// SIMATIC STEP 7 (V5.x) project Put_Get
// CPU: CPU 414-5 H (ATC-RSM)
// CPU: CPU 414-5 H (OPC-OA)
// station: P_ADR_BUS
// station: Hardware
// station: SIMATIC 400(ATC-RSM)
// station: SIMATIC 400(OPC-OA)
// station: P_ADR_BUS
// station: Hardware
// program: S7 Program
// program: S7 Program(1)

SYMBOL_TABLE
"Receive_DB"	DB 50	DB 50
"Send_DB"	DB 51	DB 51
"GET_DB"	DB 52	SFB 14
"PUT_DB"	DB 53	SFB 15
"CPU_Comm"	FC 1	FC 1
"CPU_Communication"	FC 199	FC 199
"ASSAP"	I 0.0	BOOL	//  (ATC) - (FieldIO4-M1)
"BOPL"	I 0.1	BOOL	//  (ATC) - (FieldIO4-M1)
"BVAP"	I 0.2	BOOL	//  (ATC) - (FieldIO4-M1)
"DVSAP"	I 0.3	BOOL	//  (ATC) - (FieldIO4-M1)
"EHFPL"	I 0.4	BOOL	//  (ATC) - (FieldIO4-M1)
"EHSO"	I 0.5	BOOL	//  (ATC) - (FieldIO4-M1)
"GDOGF"	I 0.6	BOOL	//  (ATC) - (FieldIO4-M1)
"GVRNLV"	I 0.7	BOOL	//  (ATC) - (FieldIO4-M1)
"HPDVC"	I 1.0	BOOL	//  (ATC) - (FieldIO4-M1)
"HPDVO"	I 1.1	BOOL	//  (ATC) - (FieldIO4-M1)
"MBCSU"	I 1.2	BOOL	//  (ATC) - (FieldIO4-M1)
"MELIT"	I 1.3	BOOL	//  (ATC) - (FieldIO4-M1)
"MVHPIT"	I 1.4	BOOL	//  (ATC) - (FieldIO4-M1)
"OEPIT"	I 1.5	BOOL	//  (ATC) - (FieldIO4-M1)
"RSBC"	I 1.6	BOOL	//  (ATC) - (FieldIO4-M1)
"RSBSU"	I 1.7	BOOL	//  (ATC) - (FieldIO4-M1)
"TGE"	I 2.0	BOOL	//  (ATC) - (FieldIO5-M1)
"VRO"	I 2.1	BOOL	//  (ATC) - (FieldIO5-M1)
"VROUS"	I 2.2	BOOL	//  (ATC) - (FieldIO5-M1)
"VRSOTP"	I 2.3	BOOL	//  (ATC) - (FieldIO5-M1)
"CAB4T1"	IW 512	WORD	//  (RSM) - (FieldIO4-M3)
"CNDP1"	IW 514	WORD	//  (RSM) - (FieldIO4-M3)
"FSST1"	IW 516	WORD	//  (RSM) - (FieldIO4-M3)
"B1T1"	IW 518	WORD	//  (ATC) - (FieldIO4-M3)
"B2T1"	IW 520	WORD	//  (ATC) - (FieldIO4-M3)
"B3T1"	IW 522	WORD	//  (ATC) - (FieldIO4-M3)
"B4T1"	IW 524	WORD	//  (ATC) - (FieldIO4-M3)
"B5T1"	IW 526	WORD	//  (ATC) - (FieldIO4-M3)
"B6T1"	IW 528	WORD	//  (ATC) - (FieldIO4-M4)
"RP1"	IW 530	WORD	//  (ATC) - (FieldIO4-M4)
"TBFCT1"	IW 532	WORD	//  (ATC) - (FieldIO4-M4)
"TBFLT1"	IW 534	WORD	//  (ATC) - (FieldIO4-M4)
"TBRCT1"	IW 536	WORD	//  (ATC) - (FieldIO4-M4)
"TBRLT1"	IW 538	WORD	//  (ATC) - (FieldIO4-M4)
"VB9"	IW 540	WORD	//  (ATC) - (FieldIO4-M4)
"FSMT1"	IW 542	WORD	//  (RSM) - (FieldIO4-M4)
"B7T"	IW 544	WORD	//  (ATC) - (FieldIO4-M5)
"B8T"	IW 546	WORD	//  (ATC) - (FieldIO4-M5)
"B9T"	IW 548	WORD	//  (ATC) - (FieldIO4-M5)
"B10T"	IW 550	WORD	//  (ATC) - (FieldIO4-M5)
"CAB5T1"	IW 552	WORD	//  (ATC) - (FieldIO4-M5)
"CAB5T2"	IW 554	WORD	//  (ATC) - (FieldIO4-M5)
"CASEXP"	IW 556	WORD	//  (ATC) - (FieldIO4-M5)
"DEGEN"	IW 558	WORD	//  (ATC) - (FieldIO4-M5)
"VB1"	IW 560	WORD	//  (ATC) - (FieldIO4-M6)
"VB2"	IW 562	WORD	//  (ATC) - (FieldIO4-M6)
"VB3"	IW 564	WORD	//  (ATC) - (FieldIO4-M6)
"VB4"	IW 566	WORD	//  (ATC) - (FieldIO4-M6)
"VB5"	IW 568	WORD	//  (ATC) - (FieldIO4-M6)
"VB6"	IW 570	WORD	//  (ATC) - (FieldIO4-M6)
"VB7"	IW 572	WORD	//  (ATC) - (FieldIO4-M6)
"VB8"	IW 574	WORD	//  (ATC) - (FieldIO4-M6)
"CAB4T2"	IW 576	WORD	//  (RSM) - (FieldIO5-M3)
"CNDP2"	IW 578	WORD	//  (RSM) - (FieldIO5-M3)
"FSST2"	IW 580	WORD	//  (RSM) - (FieldIO5-M3)
"B1T2"	IW 582	WORD	//  (ATC) - (FieldIO5-M3)
"B2T2"	IW 584	WORD	//  (ATC) - (FieldIO5-M3)
"B3T2"	IW 586	WORD	//  (ATC) - (FieldIO5-M3)
"B4T2"	IW 588	WORD	//  (ATC) - (FieldIO5-M3)
"B5T2"	IW 590	WORD	//  (ATC) - (FieldIO5-M3)
"B6T2"	IW 592	WORD	//  (ATC) - (FieldIO5-M4)
"RP2"	IW 594	WORD	//  (ATC) - (FieldIO5-M4)
"TBFCT2"	IW 596	WORD	//  (ATC) - (FieldIO5-M4)
"TBFLT2"	IW 598	WORD	//  (ATC) - (FieldIO5-M4)
"TBRCT2"	IW 600	WORD	//  (ATC) - (FieldIO5-M4)
"TBRLT2"	IW 602	WORD	//  (ATC) - (FieldIO5-M4)
"VB10"	IW 604	WORD	//  (ATC) - (FieldIO5-M4)
"LPGST"	IW 606	WORD	//  (RSM) - (FieldIO5-M4)
"EHFLT"	IW 608	WORD	//  (ATC) - (FieldIO5-M5)
"HPBMIDT"	IW 610	WORD	//  (ATC) - (FieldIO5-M5)
"HPCMIDT"	IW 612	WORD	//  (ATC) - (FieldIO5-M5)
"LP1GNT"	IW 614	WORD	//  (ATC) - (FieldIO5-M5)
"LP1GVT"	IW 616	WORD	//  (ATC) - (FieldIO5-M5)
"LP2GNT"	IW 618	WORD	//  (ATC) - (FieldIO5-M5)
"LP2GVT"	IW 620	WORD	//  (ATC) - (FieldIO5-M5)
"ROTECC"	IW 622	WORD	//  (ATC) - (FieldIO5-M5)
"OCIT"	IW 624	WORD	//  (RSM) - (FieldIO5-M6)
"OCOT"	IW 626	WORD	//  (RSM) - (FieldIO5-M6)
"Main Routine"	OB 1	OB 1
"OBNL_FLT"	OB 85	OB 85	// OB Not Loaded Fault
"PROG_ERR"	OB 121	OB 121	// Programming Error
"MOD_ERR"	OB 122	OB 122	// Module Access Error
"ATCALO"	Q 0.0	BOOL	//  (ATC) - (FieldIO4-M2)
"ATCASSO"	Q 0.1	BOOL	//  (ATC) - (FieldIO4-M2)
"ATCMEO"	Q 0.2	BOOL	//  (ATC) - (FieldIO4-M2)
"ATCNAO"	Q 0.3	BOOL	//  (ATC) - (FieldIO4-M2)
"ATCSMO"	Q 0.4	BOOL	//  (ATC) - (FieldIO4-M2)
"ATCTAO"	Q 0.5	BOOL	//  (ATC) - (FieldIO4-M2)
"ATCTO"	Q 0.6	BOOL	//  (ATC) - (FieldIO4-M2)
"CHPDVO"	Q 0.7	BOOL	//  (ATC) - (FieldIO4-M2)
"CRSBO"	Q 1.0	BOOL	//  (ATC) - (FieldIO4-M2)
"LPHTO"	Q 1.1	BOOL	//  (ATC) - (FieldIO4-M2)
"LPVHTO"	Q 1.2	BOOL	//  (ATC) - (FieldIO4-M2)
"WDHTO"	Q 1.3	BOOL	//  (ATC) - (FieldIO4-M2)
"WDVHTO"	Q 1.4	BOOL	//  (ATC) - (FieldIO4-M2)
"RSINV1"	Q 2.0	BOOL	//  (RSM) - (FieldIO5-M2)
"RSINV2"	Q 2.1	BOOL	//  (RSM) - (FieldIO5-M2)
"RSMON1"	Q 2.2	BOOL	//  (RSM) - (FieldIO5-M2)
"RSMON2"	Q 2.3	BOOL	//  (RSM) - (FieldIO5-M2)
"RSSENO"	Q 2.4	BOOL	//  (RSM) - (FieldIO5-M2)
"SPHLD"	Q 2.5	BOOL	//  (RSM) - (FieldIO5-M2)
"VAT (ATC-RSM)"	VAT 1	
END_SYMBOL_TABLE

FUNCTION "CPU_Communication" : VOID	// FC 199
TITLE = CPU_Comm
//Function call to read and write the CPU data
//
VERSION : 0.1
BEGIN
NETWORK
TITLE = Recieve data
      A     DB1.DBX 0.0;
      =     L 0.0;
      BLD   103;
      BLD   9;
      =     L 5.0;
      CDB;
      OPN   DI 1;
      TAR2  LD 1;
      A     L 0.0;
      =     DIX 0.0;
      L     1;
      T     DIW 2;
      L     W#16#1001;
      T     DIW 8;
      L     1;
      T     DIW 10;
      L     0;
      T     DIW 12;
      L     P#M 10.1;
      T     DID 14;
      L     W#16#1004;
      T     DIW 18;
      L     1;
      T     DIW 20;
      L     0;
      T     DIW 22;
      L     P#M 11.0;
      T     DID 24;
      L     W#16#1006;
      T     DIW 28;
      L     1;
      T     DIW 30;
      L     0;
      T     DIW 32;
      L     P#M 13.0;
      T     DID 34;
      L     W#16#1004;
      T     DIW 38;
      L     1;
      T     DIW 40;
      L     0;
      T     DIW 42;
      L     P#M 17.0;
      T     DID 44;
      L     W#16#1001;
      T     DIW 48;
      L     1;
      T     DIW 50;
      L     0;
      T     DIW 52;
      L     P#M 0.1;
      T     DID 54;
      L     W#16#1005;
      T     DIW 58;
      L     1;
      T     DIW 60;
      L     0;
      T     DIW 62;
      L     P#M 1.0;
      T     DID 64;
      L     W#16#1008;
      T     DIW 68;
      L     1;
      T     DIW 70;
      L     0;
      T     DIW 72;
      L     P#M 3.0;
      T     DID 74;
      L     W#16#1004;
      T     DIW 78;
      L     1;
      T     DIW 80;
      L     0;
      T     DIW 82;
      L     P#M 7.0;
      T     DID 84;
      LAR2  P#DBX 0.0;
      UC    SFB 14;
      LAR2  LD 1;
      A     DIX 4.0;
      OPN   DI 1;
      =     DIX 4.0;
      OPN   DI 1;
      A     DIX 4.1;
      OPN   DI 1;
      =     DIX 4.1;
      OPN   DI 1;
      L     DIW 6;
      OPN   DI 1;
      T     DIW 6;
      OPN   DI 1;
      CDB;
      BLD   10;
      NOP   0;
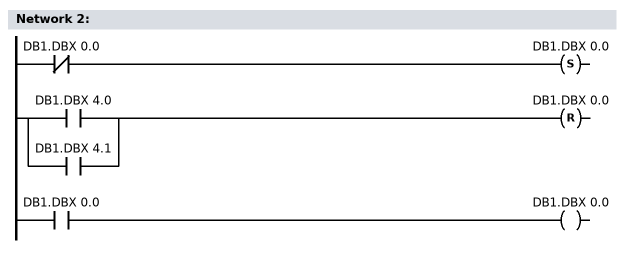
NETWORK
TITLE =
      AN    DB1.DBX 0.0;
      S     DB1.DBX 0.0;
      A(;
      O     DB1.DBX 4.0;
      O     DB1.DBX 4.1;
      );
      R     DB1.DBX 0.0;
      A     DB1.DBX 0.0;
      =     DB1.DBX 0.0;
END_FUNCTION

DATA_BLOCK "Receive_DB"	// DB 50
VERSION : 0.1
  STRUCT
   DB_VAR : INT ;	//Temporary placeholder variable
  END_STRUCT ;	
BEGIN
END_DATA_BLOCK

DATA_BLOCK "Send_DB"	// DB 51
VERSION : 0.1
  STRUCT
   DB_VAR : INT ;	//Temporary placeholder variable
  END_STRUCT ;	
BEGIN
END_DATA_BLOCK

DATA_BLOCK "GET_DB"	// DB 52
AUTHOR : SIMATIC
FAMILY : COM_FUNC
VERSION : 0.1
SFB 14
BEGIN
END_DATA_BLOCK

DATA_BLOCK "PUT_DB"	// DB 53
AUTHOR : SIMATIC
FAMILY : COM_FUNC
VERSION : 0.1
SFB 15
BEGIN
END_DATA_BLOCK

ORGANIZATION_BLOCK "Main Routine"	// OB 1
TITLE = "Main Program Sweep (Cycle)"
VERSION : 0.1
VAR_TEMP
  OB1_EV_CLASS : BYTE ;	//Bits 0-3 = 1 (Coming event), Bits 4-7 = 1 (Event class 1)
  OB1_SCAN_1 : BYTE ;	//1 (Cold restart scan 1 of OB 1), 3 (Scan 2-n of OB 1)
  OB1_PRIORITY : BYTE ;	//Priority of OB Execution
  OB1_OB_NUMBR : BYTE ;	//1 (Organization block 1, OB1)
  OB1_RESERVED_1 : BYTE ;	//Reserved for system
  OB1_RESERVED_2 : BYTE ;	//Reserved for system
  OB1_PREV_CYCLE : INT ;	//Cycle time of previous OB1 scan (milliseconds)
  OB1_MIN_CYCLE : INT ;	//Minimum cycle time of OB1 (milliseconds)
  OB1_MAX_CYCLE : INT ;	//Maximum cycle time of OB1 (milliseconds)
  OB1_DATE_TIME : DATE_AND_TIME ;	//Date and time OB1 started
END_VAR
BEGIN
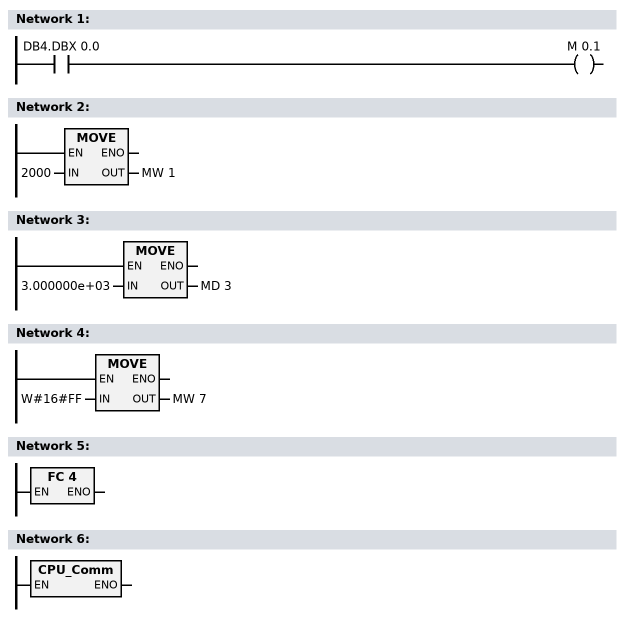
NETWORK
TITLE =
      A     DB4.DBX 0.0;
      =     M 0.1;
NETWORK
TITLE =
      L     2000;
      T     MW 1;
      NOP   0;
NETWORK
TITLE =
      L     3.000000e+03;
      T     MD 3;
      NOP   0;
NETWORK
TITLE =
      L     W#16#FF;
      T     MW 7;
      NOP   0;
NETWORK
TITLE =
      CALL  FC 4;
      NOP   0;
NETWORK
TITLE =
      CALL  "CPU_Comm";
      NOP   0;
END_ORGANIZATION_BLOCK

ORGANIZATION_BLOCK "OBNL_FLT"	// OB 85
TITLE = "Organization Block (OB) Not Loaded Fault"
VERSION : 0.1
VAR_TEMP
  OB85_EV_CLASS : BYTE ;	//16#35 Event class 3
  OB85_FLT_ID : BYTE ;	//16#XX, Fault identification code
  OB85_PRIORITY : BYTE ;	//Priority of OB Execution
  OB85_OB_NUMBR : BYTE ;	//85 (Organization block 85, OB85)
  OB85_RESERVED_1 : BYTE ;	//Reserved for system
  OB85_RESERVED_2 : BYTE ;	//Reserved for system
  OB85_RESERVED_3 : INT ;	//Reserved for system
  OB85_ERR_EV_CLASS : BYTE ;	//Class of event causing error
  OB85_ERR_EV_NUM : BYTE ;	//Number of event causing error
  OB85_OB_PRIOR : BYTE ;	//Priority of OB causing error
  OB85_OB_NUM : BYTE ;	//Number of OB causing error
  OB85_DATE_TIME : DATE_AND_TIME ;	//Date and time OB85 started
END_VAR
BEGIN
// (block stored without names or comments; labels and parameter names are numbered)
END_ORGANIZATION_BLOCK

ORGANIZATION_BLOCK "PROG_ERR"	// OB 121
TITLE = "Programming Error"
VERSION : 0.1
VAR_TEMP
  OB121_EV_CLASS : BYTE ;	//16#25, Event class 2, Entering event state, Internal fault event
  OB121_SW_FLT : BYTE ;	//16#XX Software programming fault
  OB121_PRIORITY : BYTE ;	//Priority of OB Execution
  OB121_OB_NUMBR : BYTE ;	//121 (Organization block 121, OB121)
  OB121_BLK_TYPE : BYTE ;	//16#88/8A/8B/8C/8E Type of block fault occured in
  OB121_RESERVED_1 : BYTE ;	//Reserved for system
  OB121_FLT_REG : WORD ;	//16#XX Specific register that caused fault
  OB121_BLK_NUM : WORD ;	//Number of block that programming fault occured in
  OB121_PRG_ADDR : WORD ;	//Address in block where programming fault occured
  OB121_DATE_TIME : DATE_AND_TIME ;	//Date and time OB121 started
END_VAR
BEGIN
// (block stored without names or comments; labels and parameter names are numbered)
END_ORGANIZATION_BLOCK

ORGANIZATION_BLOCK "MOD_ERR"	// OB 122
TITLE = "Module Access Error"
VERSION : 0.1
VAR_TEMP
  OB122_EV_CLASS : BYTE ;	//16#29, Event class 2, Entering event state, Internal fault event
  OB122_SW_FLT : BYTE ;	//16#XX Software error code
  OB122_PRIORITY : BYTE ;	//Priority of OB Execution
  OB122_OB_NUMBR : BYTE ;	//122 (Organization block 122, OB122)
  OB122_BLK_TYPE : BYTE ;	//16#88/8C/8E Type of block fault occured in
  OB122_MEM_AREA : BYTE ;	//Memory area where access error occured
  OB122_MEM_ADDR : WORD ;	//Memory address where access error occured
  OB122_BLK_NUM : WORD ;	//Block number in which error occured
  OB122_PRG_ADDR : WORD ;	//Program address where error occured
  OB122_DATE_TIME : DATE_AND_TIME ;	//Date and time OB1 started
END_VAR
BEGIN
// (block stored without names or comments; labels and parameter names are numbered)
END_ORGANIZATION_BLOCK

SYMBOL_TABLE
"Constants"	DB 1	DB 1
"Receive_DB"	DB 3	DB 3
"Send_DB"	DB 4	DB 4
"DB_to_Memory"	FC 3	FC 3
"Memory_to_DB"	FC 4	FC 4
"ASL1"	I 0.0	BOOL	// Auto Stop Latched # 1 (OPC) - (FieldIO1-M1)
"BR1"	I 0.1	BOOL	//  (OPC) - (FieldIO1-M1)
"INFV1"	I 0.2	BOOL	//  (OPC) - (FieldIO1-M1)
"TGRB1"	I 0.3	BOOL	//  (OPC) - (FieldIO1-M1)
"CSVBP"	I 0.4	BOOL	//  (OPC) - (FieldIO1-M1)
"CSVPB"	I 0.5	BOOL	//  (OPC) - (FieldIO1-M1)
"LCHPB"	I 0.6	BOOL	//  (OPC) - (FieldIO1-M1)
"LTPB"	I 0.7	BOOL	//  (OPC) - (FieldIO1-M1)
"OSVPB"	I 1.0	BOOL	//  (OPC) - (FieldIO1-M1)
"TMPB"	I 1.1	BOOL	//  (OPC) - (FieldIO1-M1)
"OPCT"	I 1.2	BOOL	//  (OPC) - (FieldIO1-M1)
"OST"	I 1.3	BOOL	//  (OPC) - (FieldIO1-M1)
"ADSDN"	I 2.0	BOOL	//  (OA) - (FieldIO1-M2)
"ADSPERM"	I 2.1	BOOL	//  (OA) - (FieldIO1-M2)
"ADSUP"	I 2.2	BOOL	//  (OA) - (FieldIO1-M2)
"VPLDN"	I 2.3	BOOL	//  (OA) - (FieldIO1-M2)
"VPLPERM"	I 2.4	BOOL	//  (OA) - (FieldIO1-M2)
"VPLUP"	I 2.5	BOOL	//  (OA) - (FieldIO1-M2)
"ASDN"	I 2.6	BOOL	//  (OA) - (FieldIO1-M2)
"ASPERM"	I 2.7	BOOL	//  (OA) - (FieldIO1-M2)
"ASUP"	I 3.0	BOOL	//  (OA) - (FieldIO1-M2)
"CDLPERM"	I 3.1	BOOL	//  (OA) - (FieldIO1-M2)
"FL13PRI"	I 3.2	BOOL	//  (OA) - (FieldIO1-M2)
"FL13STY"	I 3.3	BOOL	//  (OA) - (FieldIO1-M2)
"FLOACPRI"	I 3.4	BOOL	//  (OA) - (FieldIO1-M2)
"FLOACSTY"	I 3.5	BOOL	//  (OA) - (FieldIO1-M2)
"FLOPCPRI"	I 3.6	BOOL	//  (OA) - (FieldIO1-M2)
"FLOPCSTY"	I 3.7	BOOL	//  (OA) - (FieldIO1-M2)
"ASL2"	I 4.0	BOOL	//  (OPC) - (FieldIO2-M1)
"BR2"	I 4.1	BOOL	//  (OPC) - (FieldIO2-M1)
"INFV2"	I 4.2	BOOL	//  (OPC) - (FieldIO2-M1)
"TGRB2"	I 4.3	BOOL	//  (OPC) - (FieldIO2-M1)
"IV1CL"	I 6.0	BOOL	//  (OA) - (FieldIO2-M2)
"IV1OP"	I 6.1	BOOL	//  (OA) - (FieldIO2-M2)
"IV2CL"	I 6.2	BOOL	//  (OA) - (FieldIO2-M2)
"IV2OP"	I 6.3	BOOL	//  (OA) - (FieldIO2-M2)
"IV3CL"	I 6.4	BOOL	//  (OA) - (FieldIO2-M2)
"IV3OP"	I 6.5	BOOL	//  (OA) - (FieldIO2-M2)
"IV4CL"	I 6.6	BOOL	//  (OA) - (FieldIO2-M2)
"IV4OP"	I 6.7	BOOL	//  (OA) - (FieldIO2-M2)
"RV1CL"	I 7.0	BOOL	//  (OA) - (FieldIO2-M2)
"RV1OP"	I 7.1	BOOL	//  (OA) - (FieldIO2-M2)
"RV2CL"	I 7.2	BOOL	//  (OA) - (FieldIO2-M2)
"RV2OP"	I 7.3	BOOL	//  (OA) - (FieldIO2-M2)
"RV3CL"	I 7.4	BOOL	//  (OA) - (FieldIO2-M2)
"RV3OP"	I 7.5	BOOL	//  (OA) - (FieldIO2-M2)
"RV4CL"	I 7.6	BOOL	//  (OA) - (FieldIO2-M2)
"RV4OP"	I 7.7	BOOL	//  (OA) - (FieldIO2-M2)
"ASL3"	I 8.0	BOOL	//  (OPC) - (FieldIO3-M1)
"BR3"	I 8.1	BOOL	//  (OPC) - (FieldIO3-M1)
"INFV3"	I 8.2	BOOL	//  (OPC) - (FieldIO3-M1)
"TGRB3"	I 8.3	BOOL	//  (OPC) - (FieldIO3-M1)
"MSVLC"	I 8.4	BOOL	//  (OPC) - (FieldIO3-M1)
"MSVLO"	I 8.5	BOOL	//  (OPC) - (FieldIO3-M1)
"MSVRC"	I 8.6	BOOL	//  (OPC) - (FieldIO3-M1)
"MSVRO"	I 8.7	BOOL	//  (OPC) - (FieldIO3-M1)
"CI0284"	I 9.0	BOOL	//  (OPC) - (FieldIO3-M1)
"SRVOIN"	I 9.1	BOOL	//  (OPC) - (FieldIO3-M1)
"BCIV"	I 9.2	BOOL	//  (OPC) - (FieldIO3-M1)
"HOLDLOAD"	I 10.0	BOOL	//  (OA) - (FieldIO3-M2)
"REJIMP"	I 10.1	BOOL	//  (OA) - (FieldIO3-M2)
"REJMW"	I 10.2	BOOL	//  (OA) - (FieldIO3-M2)
"RESETADS"	I 10.3	BOOL	//  (OA) - (FieldIO3-M2)
"MWA"	IW 512	WORD	//  (OPC) - (FieldIO1-M5)
"OPSA"	IW 514	WORD	//  (OPC) - (FieldIO1-M5)
"OPXA"	IW 516	WORD	//  (OPC) - (FieldIO1-M5)
"TPA"	IW 518	WORD	//  (OPC) - (FieldIO1-M5)
"PIA"	IW 520	WORD	//  (OA) - (FieldIO1-M5)
"GSH1"	IW 522	WORD	//  (OA) - (FieldIO1-M5)
"STATCUR"	IW 524	WORD	//  (OPC) - (FieldIO1-M5)
"MWB"	IW 528	WORD	//  (OPC) - (FieldIO2-M5)
"OPSB"	IW 530	WORD	//  (OPC) - (FieldIO2-M5)
"OPXB"	IW 532	WORD	//  (OPC) - (FieldIO2-M5)
"TPB"	IW 534	WORD	//  (OPC) - (FieldIO2-M5)
"PIB"	IW 536	WORD	//  (OA) - (FieldIO2-M5)
"GSHP2"	IW 538	WORD	//  (OA) - (FieldIO2-M5)
"PLRL"	IW 540	WORD	//  (OA) - (FieldIO2-M5)
"MWC"	IW 544	WORD	//  (OPC) - (FieldIO3-M5)
"OPSC"	IW 546	WORD	//  (OPC) - (FieldIO3-M5)
"OPXC"	IW 548	WORD	//  (OPC) - (FieldIO3-M5)
"TPC"	IW 550	WORD	//  (OPC) - (FieldIO3-M5)
"PIC"	IW 552	WORD	//  (OA) - (FieldIO3-M5)
"MVAR"	IW 554	WORD	//  (OPC) - (FieldIO3-M5)
"AA"	M 10.1	BOOL
"CC"	MD 13	REAL
"BB"	MW 11	INT
"DD"	MW 17	WORD
"Main Program"	OB 1	OB 1
"OBNL_FLT"	OB 85	OB 85	// OB Not Loaded Fault
"PROG_ERR"	OB 121	OB 121	// Programming Error
"MOD_ERR"	OB 122	OB 122	// Module Access Error
"TM1"	Q 0.0	BOOL	//  (OPC) - (FieldIO1-M3)
"LATCH1"	Q 0.1	BOOL	//  (OPC) - (FieldIO1-M3)
"TTRIP1"	Q 0.2	BOOL	//  (OPC) - (FieldIO1-M3)
"PSMN1"	Q 0.3	BOOL	//  (OPC) - (FieldIO1-M3)
"OSPD1"	Q 0.4	BOOL	//  (OPC) - (FieldIO1-M3)
"SRVOOUT1"	Q 0.5	BOOL	//  (OPC) - (FieldIO1-M3)
"OPCO1"	Q 0.6	BOOL	//  (OPC) - (FieldIO1-M3)
"OPMN1"	Q 0.7	BOOL	//  (OPC) - (FieldIO1-M3)
"MRBC"	Q 1.0	BOOL	//  (OPC) - (FieldIO1-M3)
"MRBRC"	Q 1.1	BOOL	//  (OPC) - (FieldIO1-M3)
"MVPMAN"	Q 1.2	BOOL	//  (OPC) - (FieldIO1-M3)
"ASLNLT"	Q 1.3	BOOL	//  (OPC) - (FieldIO1-M3)
"ASLT"	Q 1.4	BOOL	//  (OPC) - (FieldIO1-M3)
"GVCL"	Q 1.5	BOOL	//  (OPC) - (FieldIO1-M3)
"LT"	Q 1.6	BOOL	//  (OPC) - (FieldIO1-M3)
"ADS1"	Q 2.0	BOOL	//  (OA) - (FieldIO1-M4)
"AS1"	Q 2.1	BOOL	//  (OA) - (FieldIO1-M4)
"BRCTT1"	Q 2.2	BOOL	//  (OA) - (FieldIO1-M4)
"DMWFL1"	Q 2.3	BOOL	//  (OA) - (FieldIO1-M4)
"HLLL1"	Q 2.4	BOOL	//  (OA) - (FieldIO1-M4)
"IPI1"	Q 2.5	BOOL	//  (OA) - (FieldIO1-M4)
"LLLL1"	Q 2.6	BOOL	//  (OA) - (FieldIO1-M4)
"LOWFRQ1"	Q 2.7	BOOL	//  (OA) - (FieldIO1-M4)
"MWFAIL1"	Q 3.0	BOOL	//  (OA) - (FieldIO1-M4)
"MWI1"	Q 3.1	BOOL	//  (OA) - (FieldIO1-M4)
"OA1"	Q 3.2	BOOL	//  (OA) - (FieldIO1-M4)
"OPXFAIL1"	Q 3.3	BOOL	//  (OA) - (FieldIO1-M4)
"PIFAIL1"	Q 3.4	BOOL	//  (OA) - (FieldIO1-M4)
"PLRLL1"	Q 3.5	BOOL	//  (OA) - (FieldIO1-M4)
"SPI1"	Q 3.6	BOOL	//  (OA) - (FieldIO1-M4)
"TPFAIL1"	Q 3.7	BOOL	//  (OA) - (FieldIO1-M4)
"TM2"	Q 4.0	BOOL	//  (OPC) - (FieldIO2-M3)
"LATCH2"	Q 4.1	BOOL	//  (OPC) - (FieldIO2-M3)
"TTRIP2"	Q 4.2	BOOL	//  (OPC) - (FieldIO2-M3)
"PSMN2"	Q 4.3	BOOL	//  (OPC) - (FieldIO2-M3)
"OSPD2"	Q 4.4	BOOL	//  (OPC) - (FieldIO2-M3)
"SRVOOUT2"	Q 4.5	BOOL	//  (OPC) - (FieldIO2-M3)
"OPCO2"	Q 4.6	BOOL	//  (OPC) - (FieldIO2-M3)
"OPMN2"	Q 4.7	BOOL	//  (OPC) - (FieldIO2-M3)
"MWLT"	Q 5.0	BOOL	//  (OPC) - (FieldIO2-M3)
"OPCMONLT"	Q 5.1	BOOL	//  (OPC) - (FieldIO2-M3)
"PFAILT"	Q 5.2	BOOL	//  (OPC) - (FieldIO2-M3)
"RPMLT"	Q 5.3	BOOL	//  (OPC) - (FieldIO2-M3)
"STROBE"	Q 5.4	BOOL	//  (OPC) - (FieldIO2-M3)
"TMLT"	Q 5.5	BOOL	//  (OPC) - (FieldIO2-M3)
"TMLT1"	Q 5.6	BOOL	//  (OPC) - (FieldIO2-M3)
"TVCL"	Q 5.7	BOOL	//  (OPC) - (FieldIO2-M3)
"ADS2"	Q 6.0	BOOL	//  (OA) - (FieldIO2-M4)
"AS2"	Q 6.1	BOOL	//  (OA) - (FieldIO2-M4)
"BRCTT2"	Q 6.2	BOOL	//  (OA) - (FieldIO2-M4)
"DMWFL2"	Q 6.3	BOOL	//  (OA) - (FieldIO2-M4)
"HLLL2"	Q 6.4	BOOL	//  (OA) - (FieldIO2-M4)
"IPI2"	Q 6.5	BOOL	//  (OA) - (FieldIO2-M4)
"LLLL2"	Q 6.6	BOOL	//  (OA) - (FieldIO2-M4)
"LOWFRQ2"	Q 6.7	BOOL	//  (OA) - (FieldIO2-M4)
"MWFAIL2"	Q 7.0	BOOL	//  (OA) - (FieldIO2-M4)
"MWI2"	Q 7.1	BOOL	//  (OA) - (FieldIO2-M4)
"OA2"	Q 7.2	BOOL	//  (OA) - (FieldIO2-M4)
"OPXFAIL2"	Q 7.3	BOOL	//  (OA) - (FieldIO2-M4)
"PIFAIL2"	Q 7.4	BOOL	//  (OA) - (FieldIO2-M4)
"PLRLL2"	Q 7.5	BOOL	//  (OA) - (FieldIO2-M4)
"SPI2"	Q 7.6	BOOL	//  (OA) - (FieldIO2-M4)
"TPFAIL2"	Q 7.7	BOOL	//  (OA) - (FieldIO2-M4)
"TM3"	Q 8.0	BOOL	//  (OPC) - (FieldIO3-M3)
"OPCO"	Q 8.1	BOOL	//  (OPC) - (FieldIO3-M3)
"SRVOLT"	Q 8.2	BOOL	//  (OPC) - (FieldIO3-M3)
"ASL"	Q 8.3	BOOL	//  (OPC) - (FieldIO3-M3)
"ASLDOR"	Q 8.4	BOOL	//  (OPC) - (FieldIO3-M3)
"CIV"	Q 8.5	BOOL	//  (OPC) - (FieldIO3-M3)
"EIVN"	Q 8.6	BOOL	//  (OPC) - (FieldIO3-M3)
"CIV1"	Q 8.7	BOOL	//  (OPC) - (FieldIO3-M3)
"CIV2"	Q 9.0	BOOL	//  (OPC) - (FieldIO3-M3)
"CIV3"	Q 9.1	BOOL	//  (OPC) - (FieldIO3-M3)
"CIV4"	Q 9.2	BOOL	//  (OPC) - (FieldIO3-M3)
"MSTPVL"	Q 9.3	BOOL	//  (OPC) - (FieldIO3-M3)
"MSTPVR"	Q 9.4	BOOL	//  (OPC) - (FieldIO3-M3)
"MTPRBMVP"	Q 9.5	BOOL	//  (OPC) - (FieldIO3-M3)
"TGRB"	Q 9.6	BOOL	//  (OPC) - (FieldIO3-M3)
"MANNAUTO"	Q 9.7	BOOL	//  (OA) - (FieldIO3-M3)
"HLLI"	Q 10.0	BOOL	//  (OA) - (FieldIO3-M4)
"LFRQO"	Q 10.1	BOOL	//  (OA) - (FieldIO3-M4)
"LLDO"	Q 10.2	BOOL	//  (OA) - (FieldIO3-M4)
"LLLI"	Q 10.3	BOOL	//  (OA) - (FieldIO3-M4)
"MOTO"	Q 10.4	BOOL	//  (OA) - (FieldIO3-M4)
"RBOP"	Q 10.5	BOOL	//  (OA) - (FieldIO3-M4)
"RCLINHO"	Q 10.6	BOOL	//  (OA) - (FieldIO3-M4)
"RCRINHO"	Q 10.7	BOOL	//  (OA) - (FieldIO3-M4)
"TSTRV1"	Q 11.0	BOOL	//  (OA) - (FieldIO3-M4)
"TSTRV2"	Q 11.1	BOOL	//  (OA) - (FieldIO3-M4)
"TSTRV3"	Q 11.2	BOOL	//  (OA) - (FieldIO3-M4)
"TSTRV4"	Q 11.3	BOOL	//  (OA) - (FieldIO3-M4)
"VPLL1"	Q 11.4	BOOL	//  (OA) - (FieldIO3-M4)
"VPLL2"	Q 11.5	BOOL	//  (OA) - (FieldIO3-M4)
"WSFAIL1"	Q 11.6	BOOL	//  (OA) - (FieldIO3-M4)
"WSFAIL2"	Q 11.7	BOOL	//  (OA) - (FieldIO3-M4)
"VAT (OPC-OA)"	VAT 1	
END_SYMBOL_TABLE

FUNCTION "DB_to_Memory" : VOID	// FC 3
TITLE = DB_to_Memory
//
//To move data from DB variables to memory variables
//
AUTHOR : RJ
VERSION : 0.0
BEGIN
// body was compiled from an SCL source; compiled code not shown
END_FUNCTION

FUNCTION "Memory_to_DB" : VOID	// FC 4
TITLE = Memory_to_DB
//
//To move data from to memory variables DB variables 
//
AUTHOR : RJ
VERSION : 0.0
BEGIN
// body was compiled from an SCL source; compiled code not shown
END_FUNCTION

DATA_BLOCK "Constants"	// DB 1
VERSION : 0.1
  STRUCT
   A : BOOL  := TRUE;
   B : INT  := 1234;
   C : REAL  := 4.321000e+003;
   D : WORD  := W#16#FF;
  END_STRUCT ;	
BEGIN
END_DATA_BLOCK

DATA_BLOCK "Receive_DB"	// DB 3
TITLE = 'Receive_DB'
//
// Insert a variable for every memory variable that are to be received to partner CPU
//
//
AUTHOR : RJ
VERSION : 0.0
  STRUCT
   A : BOOL ;
   B : INT ;
   C : REAL ;
   D : WORD ;
   E : DWORD ;
  END_STRUCT ;	
BEGIN
END_DATA_BLOCK

DATA_BLOCK "Send_DB"	// DB 4
TITLE = 'Send_DB'
//
// Insert a variable for every memory variable that are to be received to partner CPU
//
//
AUTHOR : RJ
VERSION : 0.0
  STRUCT
   A : BOOL ;
   B : INT ;
   C : REAL ;
   D : WORD ;
   E : DWORD ;
  END_STRUCT ;	
BEGIN
END_DATA_BLOCK

ORGANIZATION_BLOCK "Main Program"	// OB 1
TITLE = "Main Program Sweep (Cycle)"
VERSION : 0.1
VAR_TEMP
  OB1_EV_CLASS : BYTE ;	//Bits 0-3 = 1 (Coming event), Bits 4-7 = 1 (Event class 1)
  OB1_SCAN_1 : BYTE ;	//1 (Cold restart scan 1 of OB 1), 3 (Scan 2-n of OB 1)
  OB1_PRIORITY : BYTE ;	//Priority of OB Execution
  OB1_OB_NUMBR : BYTE ;	//1 (Organization block 1, OB1)
  OB1_RESERVED_1 : BYTE ;	//Reserved for system
  OB1_RESERVED_2 : BYTE ;	//Reserved for system
  OB1_PREV_CYCLE : INT ;	//Cycle time of previous OB1 scan (milliseconds)
  OB1_MIN_CYCLE : INT ;	//Minimum cycle time of OB1 (milliseconds)
  OB1_MAX_CYCLE : INT ;	//Maximum cycle time of OB1 (milliseconds)
  OB1_DATE_TIME : DATE_AND_TIME ;	//Date and time OB1 started
END_VAR
BEGIN
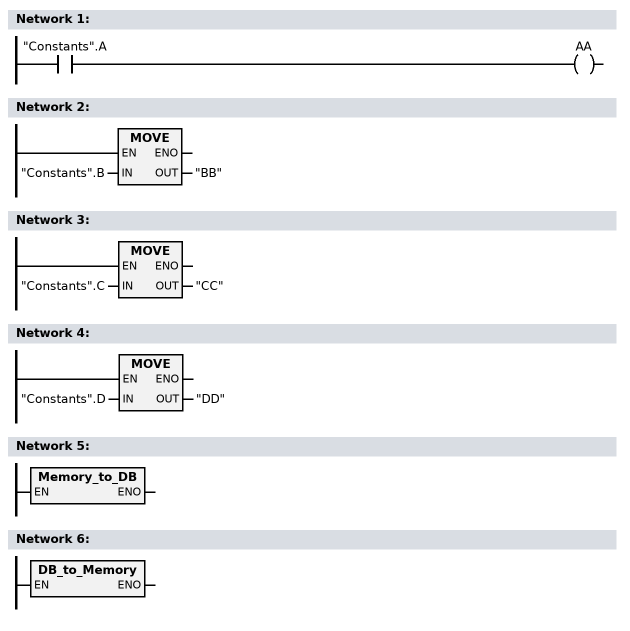
NETWORK
TITLE =
      A     "Constants".A;
      =     "AA";
NETWORK
TITLE =
      L     "Constants".B;
      T     "BB";
      NOP   0;
NETWORK
TITLE =
      L     "Constants".C;
      T     "CC";
      NOP   0;
NETWORK
TITLE =
      L     "Constants".D;
      T     "DD";
      NOP   0;
NETWORK
TITLE =
      CALL  "Memory_to_DB";
      NOP   0;
NETWORK
TITLE =
      CALL  "DB_to_Memory";
      NOP   0;
END_ORGANIZATION_BLOCK

ORGANIZATION_BLOCK "OBNL_FLT"	// OB 85
TITLE = "Organization Block (OB) Not Loaded Fault"
VERSION : 0.1
VAR_TEMP
  OB85_EV_CLASS : BYTE ;	//16#35 Event class 3
  OB85_FLT_ID : BYTE ;	//16#XX, Fault identification code
  OB85_PRIORITY : BYTE ;	//Priority of OB Execution
  OB85_OB_NUMBR : BYTE ;	//85 (Organization block 85, OB85)
  OB85_RESERVED_1 : BYTE ;	//Reserved for system
  OB85_RESERVED_2 : BYTE ;	//Reserved for system
  OB85_RESERVED_3 : INT ;	//Reserved for system
  OB85_ERR_EV_CLASS : BYTE ;	//Class of event causing error
  OB85_ERR_EV_NUM : BYTE ;	//Number of event causing error
  OB85_OB_PRIOR : BYTE ;	//Priority of OB causing error
  OB85_OB_NUM : BYTE ;	//Number of OB causing error
  OB85_DATE_TIME : DATE_AND_TIME ;	//Date and time OB85 started
END_VAR
BEGIN
// (block stored without names or comments; labels and parameter names are numbered)
END_ORGANIZATION_BLOCK

ORGANIZATION_BLOCK "PROG_ERR"	// OB 121
TITLE = "Programming Error"
VERSION : 0.1
VAR_TEMP
  OB121_EV_CLASS : BYTE ;	//16#25, Event class 2, Entering event state, Internal fault event
  OB121_SW_FLT : BYTE ;	//16#XX Software programming fault
  OB121_PRIORITY : BYTE ;	//Priority of OB Execution
  OB121_OB_NUMBR : BYTE ;	//121 (Organization block 121, OB121)
  OB121_BLK_TYPE : BYTE ;	//16#88/8A/8B/8C/8E Type of block fault occured in
  OB121_RESERVED_1 : BYTE ;	//Reserved for system
  OB121_FLT_REG : WORD ;	//16#XX Specific register that caused fault
  OB121_BLK_NUM : WORD ;	//Number of block that programming fault occured in
  OB121_PRG_ADDR : WORD ;	//Address in block where programming fault occured
  OB121_DATE_TIME : DATE_AND_TIME ;	//Date and time OB121 started
END_VAR
BEGIN
// (block stored without names or comments; labels and parameter names are numbered)
END_ORGANIZATION_BLOCK

ORGANIZATION_BLOCK "MOD_ERR"	// OB 122
TITLE = "Module Access Error"
VERSION : 0.1
VAR_TEMP
  OB122_EV_CLASS : BYTE ;	//16#29, Event class 2, Entering event state, Internal fault event
  OB122_SW_FLT : BYTE ;	//16#XX Software error code
  OB122_PRIORITY : BYTE ;	//Priority of OB Execution
  OB122_OB_NUMBR : BYTE ;	//122 (Organization block 122, OB122)
  OB122_BLK_TYPE : BYTE ;	//16#88/8C/8E Type of block fault occured in
  OB122_MEM_AREA : BYTE ;	//Memory area where access error occured
  OB122_MEM_ADDR : WORD ;	//Memory address where access error occured
  OB122_BLK_NUM : WORD ;	//Block number in which error occured
  OB122_PRG_ADDR : WORD ;	//Program address where error occured
  OB122_DATE_TIME : DATE_AND_TIME ;	//Date and time OB1 started
END_VAR
BEGIN
// (block stored without names or comments; labels and parameter names are numbered)
END_ORGANIZATION_BLOCK
